FUNCTION_BLOCK TON_Wrapper implements I_TON
VAR
    {attribute 'hide'} _ton : TON;
    {attribute 'hide'} _q 	: BOOL;
   	{attribute 'hide'} _et 	: TIME;
END_VAR

 
METHOD Call : BOOL
VAR_INPUT
	IN	: BOOL;
	PT	: TIME;
END_VAR
VAR_OUTPUT
	Q 	: BOOL;
	ET 	: TIME;
END_VAR

_ton(IN := IN, PT := PT);
Q := _ton.Q;
ET := _ton.ET;
END_METHOD

END_FUNCTION_BLOCK

(* stored: Version 1.1.0.1, ProductVersion 3.1.4024.9
   POU TON_Wrapper: Id {d29dc3bb-fcc7-4177-b77e-d087a4341de6}, SpecialFunc None
   Method Call: Id {79924cb8-d06d-4c5a-9852-6be0b3cb3d4c} *)
